TYPE ST_MotionlinxAI_Axis_Status :
	STRUCT
		Extended   : BOOL;
		Retracted  : BOOL;
		Extending  : BOOL;
		Retracting : BOOL;
	END_STRUCT
END_TYPE

(* stored: Version 1.1.0.1, ProductVersion 3.1.4024.15
   DUT ST_MotionlinxAI_Axis_Status: Id {b7396a8d-b695-4c2f-8e27-42276537eaba} *)
